Universal Robots PolyScope program: tip_change_JF.urp

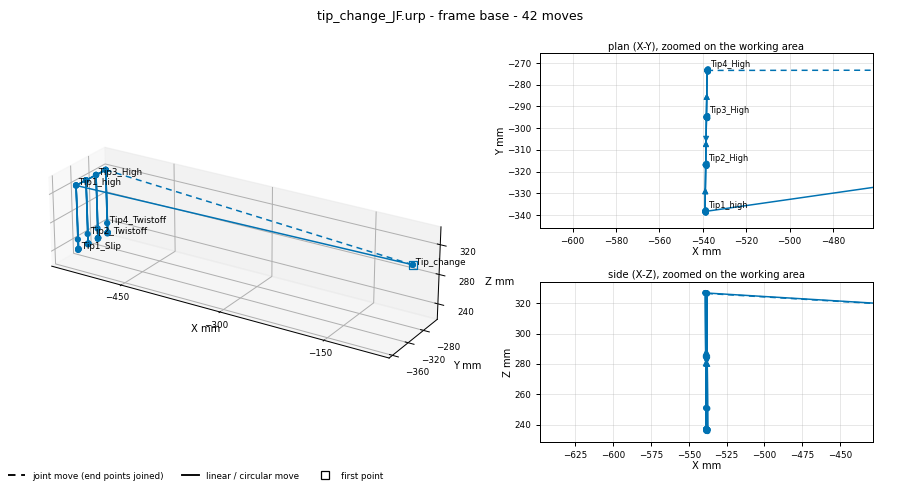
[picture p0: tool path of tip_change_JF.urp in frame base, 42 of 42 moves have a stored position in this frame; points joined in program order, loops and branches not executed]
Program tip_change_JF (installation=default directory=/programs/usbdisk/Ur-Program/Tip_change createdIn=3.10.1.76190 lastSavedIn=3.10.1.76190 robotSerialNumber=2018359886)
Calibrated DH parameters: a=[-0.000111, -0.180064, -0.391564, 0.000025, 0.000035, 0]; d=[0.089308, 162.079685, -160.155007, -1.814221, 0.094754, 0.082578]; alpha=[1.569707, -0.002379, 0.010338, 1.570474, -1.569894, 0]; deltaTheta=[0.000021, -1.133914, 1.184629, -0.050828, 0.000017, 0.000075]
Robot Program (runOnlyOnce=false)
  MoveJ speed 60 deg/s, acceleration 80 deg/s^2 (useActiveTCP=false) tcp=TCP_Tool1
    Waypoint Tip_change: TCP in base x=-81.571 y=-272.848 z=299.256 mm, rx=0 ry=0.0001 rz=-1.545 rad; joints [-70.556, -50.466, -101.854, -104.569, 84.569, 123.199] deg; flange x=-49.667 y=-215.719 z=542.134 mm, rx=2.3303 ry=1.8037 rz=-0.2542 rad
  Set NoAction tcp=TCP_Tool1
  'skipping tip 0-> No tool on robot'
  If Old_tip≟3
    MoveL speed 250 mm/s, acceleration 1200 mm/s^2 (useActiveTCP=false) tcp=TCP_Tool1; feature=Joint_6_name
      Waypoint Tip1_high: TCP in base x=-538.968 y=-338.378 z=326.942 mm, rx=-0.0068 ry=0.0085 rz=3.1265 rad; joints [-131.445, -107.957, -50.262, -104.103, 80.885, 154.293] deg; pose in feature x=57.214 y=-30.744 z=76.425 mm, rx=0 ry=0.0001 rz=-2.0641 rad; flange x=-490.354 y=-366.84 z=572.437 mm, rx=3.0721 ry=-0.4473 rz=-0.3327 rad
      Waypoint Tip1_Slip: TCP in base x=-538.568 y=-337.869 z=236.939 mm, rx=-0.0068 ry=0.0085 rz=3.1242 rad; joints [-131.488, -104.349, -68.619, -89.398, 80.899, 154.544] deg; pose in feature x=-140.414 y=-433.139 z=348.51 mm, rx=0.0255 ry=-0.0126 rz=-1.9429 rad; flange x=-490.024 y=-366.448 z=482.434 mm, rx=3.0718 ry=-0.4509 rz=-0.3328 rad
      Waypoint Tip1_Lock: TCP in base x=-538.583 y=-338.869 z=236.944 mm, rx=0.0013 ry=-0.0083 rz=-2.1118 rad; joints [-137.124, -99.221, -76.057, -82.468, 93.606, 89.965] deg; pose in feature x=-139.482 y=-433.5 z=348.531 mm, rx=0.0139 ry=-0.0208 rz=-0.8958 rad; flange x=-488.924 y=-309.541 z=482.128 mm, rx=2.7896 ry=1.107 rz=-0.2715 rad
      Waypoint Tip1_Twistoff: TCP in base x=-538.643 y=-338.793 z=250.944 mm, rx=-0.0027 ry=-0.0068 rz=-1.059 rad; joints [-143.816, -105.991, -63.242, -98.539, 103.242, 22.663] deg; pose in feature x=-0.02 y=-0.021 z=11.036 mm, rx=-0.0001 ry=0 rz=1.0527 rad; flange x=-538.901 y=-279.541 z=495.751 mm, rx=1.814 ry=2.3069 rz=-0.1444 rad
      Waypoint Tip1_high: TCP in base x=-538.968 y=-338.378 z=326.942 mm, rx=-0.0068 ry=0.0085 rz=3.1265 rad; joints [-131.445, -107.957, -50.262, -104.103, 80.885, 154.293] deg; pose in feature x=57.214 y=-30.744 z=76.425 mm, rx=0 ry=0.0001 rz=-2.0641 rad; flange x=-490.354 y=-366.84 z=572.437 mm, rx=3.0721 ry=-0.4473 rz=-0.3327 rad
    SuppressedNode
      MoveL speed 250 mm/s, acceleration 1200 mm/s^2 (useActiveTCP=false) tcp=TCP_Tool1; feature=Joint_6_name
        Waypoint Tip1_high: TCP in base x=-537.538 y=-337.809 z=326.901 mm, rx=0.0003 ry=0.0002 rz=-1.5826 rad; joints [-130.16, -106.928, -52.243, -102.922, -281.606, 155.501] deg; pose in feature x=0.604 y=0.279 z=0.912 mm, rx=0 ry=0.0001 rz=0.0099 rad; flange x=-481.613 y=-371.883 z=569.759 mm, rx=3.08 ry=-0.4512 rz=-0.394 rad
        Waypoint Tip1_press: TCP in base x=-537.53 y=-337.783 z=237.901 mm, rx=0.0003 ry=0 rz=-0.5354 rad; joints [-136.639, -97.589, -78.691, -79.527, -267.198, 90.394] deg; pose in feature x=-0.011 y=0.014 z=-89.017 mm, rx=0 ry=-0.0001 rz=1.0471 rad; flange x=-480.131 y=-306.405 z=480.779 mm, rx=2.7834 ry=1.1057 rz=-0.3248 rad
        Waypoint Tip1_Lock: TCP in base x=-537.531 y=-337.784 z=239.901 mm, rx=0.0003 ry=0 rz=-0.5354 rad; joints [-136.638, -97.608, -78.375, -79.823, -267.198, 90.392] deg; pose in feature x=-0.011 y=0.014 z=-87.017 mm, rx=0 ry=0 rz=1.0471 rad; flange x=-480.132 y=-306.408 z=482.779 mm, rx=2.7834 ry=1.1057 rz=-0.3248 rad
        Waypoint Tip1_Slip: TCP in base x=-537.531 y=-337.783 z=238.901 mm, rx=0.0003 ry=0.0001 rz=-1.5826 rad; joints [-130.205, -103.681, -69.728, -88.707, -281.576, 155.612] deg; pose in feature x=0.094 y=0.018 z=1.031 mm, rx=-0.0001 ry=-0.0001 rz=0.0001 rad; flange x=-481.61 y=-371.853 z=481.761 mm, rx=3.0799 ry=-0.4512 rz=-0.3939 rad
        Waypoint Tip1_high: TCP in base x=-537.538 y=-337.809 z=326.901 mm, rx=0.0003 ry=0.0002 rz=-1.5826 rad; joints [-130.16, -106.928, -52.243, -102.922, -281.606, 155.501] deg; pose in feature x=0.604 y=0.279 z=0.912 mm, rx=0 ry=0.0001 rz=0.0099 rad; flange x=-481.613 y=-371.883 z=569.759 mm, rx=3.08 ry=-0.4512 rz=-0.394 rad
  If Old_tip≟4
    MoveL speed 250 mm/s, acceleration 1200 mm/s^2 (useActiveTCP=false) tcp=TCP_Tool1; feature=Joint_6_name
      Waypoint Tip2_High: TCP in base x=-538.644 y=-316.88 z=326.826 mm, rx=-0.0068 ry=0.0085 rz=3.1265 rad; joints [-132.848, -105.784, -53.248, -103.06, 81.079, 152.898] deg; pose in feature x=2.19 y=1.693 z=81.747 mm, rx=-0.0035 ry=0.0068 rz=-0.958 rad; flange x=-490.029 y=-345.343 z=572.321 mm, rx=3.0721 ry=-0.4473 rz=-0.3327 rad
      Waypoint Tip2_Slip: TCP in base x=-538.244 y=-316.372 z=236.823 mm, rx=-0.0068 ry=0.0085 rz=3.1265 rad; joints [-132.898, -102.409, -71.128, -88.573, 81.109, 153.006] deg; pose in feature x=-160.454 y=-425.366 z=348.057 mm, rx=0.0255 ry=-0.0126 rz=-1.9406 rad; flange x=-489.629 y=-344.835 z=482.318 mm, rx=3.0721 ry=-0.4473 rz=-0.3327 rad
      Waypoint Tip2_Lock: TCP in base x=-538.259 y=-317.372 z=236.828 mm, rx=0.0012 ry=-0.0083 rz=-2.1095 rad; joints [-138.801, -97.64, -77.885, -82.321, 93.99, 88.197] deg; pose in feature x=-159.522 y=-425.727 z=348.078 mm, rx=0.0138 ry=-0.0208 rz=-0.8934 rad; flange x=-488.666 y=-287.924 z=482.011 mm, rx=2.7881 ry=1.1102 rz=-0.2712 rad
      Waypoint Tip2_Twistoff: TCP in base x=-538.319 y=-317.295 z=250.828 mm, rx=-0.0027 ry=-0.0068 rz=-1.0623 rad; joints [-145.487, -104.574, -65.006, -98.529, 103.298, 21.145] deg; pose in feature x=-0.013 y=0.071 z=-74.909 mm, rx=0.0001 ry=-0.0001 rz=2.0945 rad; flange x=-538.389 y=-258.046 z=495.635 mm, rx=1.8178 ry=2.3041 rz=-0.1448 rad
      Waypoint Tip2_High: TCP in base x=-538.644 y=-316.88 z=326.826 mm, rx=-0.0068 ry=0.0085 rz=3.1265 rad; joints [-132.848, -105.784, -53.248, -103.06, 81.079, 152.898] deg; pose in feature x=2.19 y=1.693 z=81.747 mm, rx=-0.0035 ry=0.0068 rz=-0.958 rad; flange x=-490.029 y=-345.343 z=572.321 mm, rx=3.0721 ry=-0.4473 rz=-0.3327 rad
    SuppressedNode
      MoveL speed 250 mm/s, acceleration 1200 mm/s^2 (useActiveTCP=false) tcp=TCP_Tool1; feature=Joint_6_name
        Waypoint Tip2_High: TCP in base x=-537.283 y=-316.311 z=326.907 mm, rx=0.0003 ry=0.0002 rz=-1.5826 rad; joints [-131.544, -104.755, -55.177, -101.873, -281.409, 154.115] deg; pose in feature x=-21.513 y=0.011 z=-0.018 mm, rx=0 ry=0 rz=-0.0001 rad; flange x=-481.359 y=-350.384 z=569.766 mm, rx=3.08 ry=-0.4512 rz=-0.394 rad
        Waypoint Tip2_Press: TCP in base x=-537.276 y=-316.285 z=237.907 mm, rx=0.0003 ry=0 rz=-0.5354 rad; joints [-138.326, -96.017, -80.448, -79.412, -266.784, 88.762] deg; pose in feature x=-21.511 y=0.015 z=-89.018 mm, rx=0 ry=-0.0001 rz=1.0471 rad; flange x=-479.877 y=-284.907 z=480.785 mm, rx=2.7834 ry=1.1057 rz=-0.3248 rad
        Waypoint Tip2_Lock: TCP in base x=-537.276 y=-316.285 z=239.907 mm, rx=0.0003 ry=0 rz=-0.5354 rad; joints [-138.325, -96.035, -80.135, -79.708, -266.784, 88.759] deg; pose in feature x=-21.511 y=0.015 z=-87.018 mm, rx=0 ry=0 rz=1.0471 rad; flange x=-479.878 y=-284.909 z=482.785 mm, rx=2.7834 ry=1.1057 rz=-0.3248 rad
        Waypoint Tip2_Slip: TCP in base x=-537.276 y=-316.285 z=238.907 mm, rx=0.0003 ry=0.0001 rz=-1.5826 rad; joints [-131.59, -101.734, -72.212, -87.881, -281.381, 154.223] deg; pose in feature x=-21.511 y=0.015 z=-88.018 mm, rx=0.0001 ry=0 rz=-0.0001 rad; flange x=-481.356 y=-350.354 z=481.767 mm, rx=3.0799 ry=-0.4512 rz=-0.3939 rad
        Waypoint Tip2_High: TCP in base x=-537.283 y=-316.311 z=326.907 mm, rx=0.0003 ry=0.0002 rz=-1.5826 rad; joints [-131.544, -104.755, -55.177, -101.873, -281.409, 154.115] deg; pose in feature x=-21.513 y=0.011 z=-0.018 mm, rx=0 ry=0 rz=-0.0001 rad; flange x=-481.359 y=-350.384 z=569.766 mm, rx=3.08 ry=-0.4512 rz=-0.394 rad
  If Old_tip≟5
    MoveL speed 250 mm/s, acceleration 1200 mm/s^2 (useActiveTCP=false) tcp=TCP_Tool1; feature=Joint_6_name
      Waypoint Tip3_High: TCP in base x=-538.312 y=-294.883 z=326.707 mm, rx=-0.0068 ry=0.0085 rz=3.1265 rad; joints [-134.359, -103.714, -56.012, -102.124, 81.293, 151.396] deg; pose in feature x=13.69 y=-3.755 z=-38.348 mm, rx=-0.1637 ry=0.1574 rz=-0.0025 rad; flange x=-489.697 y=-323.346 z=572.202 mm, rx=3.0721 ry=-0.4473 rz=-0.3327 rad
      Waypoint Tip3_Slip: TCP in base x=-537.912 y=-294.375 z=236.704 mm, rx=-0.0068 ry=0.0085 rz=3.1265 rad; joints [-134.411, -100.547, -73.471, -87.848, 81.321, 151.499] deg; pose in feature x=-180.961 y=-417.412 z=347.593 mm, rx=0.0255 ry=-0.0126 rz=-1.9406 rad; flange x=-489.297 y=-322.838 z=482.199 mm, rx=3.0721 ry=-0.4473 rz=-0.3327 rad
      Waypoint Tip3_Lock: TCP in base x=-537.927 y=-295.375 z=236.709 mm, rx=0.0012 ry=-0.0083 rz=-2.1095 rad; joints [-140.58, -96.119, -79.595, -82.242, 94.365, 86.458] deg; pose in feature x=-180.029 y=-417.773 z=347.614 mm, rx=0.0138 ry=-0.0208 rz=-0.8934 rad; flange x=-488.334 y=-265.927 z=481.892 mm, rx=2.7881 ry=1.1102 rz=-0.2712 rad
      Waypoint Tip3_Twistoff: TCP in base x=-537.987 y=-295.298 z=250.709 mm, rx=-0.0027 ry=-0.0068 rz=-1.0623 rad; joints [-147.274, -103.276, -66.568, -98.672, 103.353, 19.316] deg; pose in feature x=-1.767 y=-0.914 z=5.336 mm, rx=0 ry=0 rz=1.0005 rad; flange x=-538.057 y=-236.049 z=495.517 mm, rx=1.8178 ry=2.3041 rz=-0.1448 rad
      Waypoint Tip3_High: TCP in base x=-538.312 y=-294.883 z=326.707 mm, rx=-0.0068 ry=0.0085 rz=3.1265 rad; joints [-134.359, -103.714, -56.012, -102.124, 81.293, 151.396] deg; pose in feature x=13.69 y=-3.755 z=-38.348 mm, rx=-0.1637 ry=0.1574 rz=-0.0025 rad; flange x=-489.697 y=-323.346 z=572.202 mm, rx=3.0721 ry=-0.4473 rz=-0.3327 rad
    SuppressedNode
      MoveL speed 250 mm/s, acceleration 1200 mm/s^2 (useActiveTCP=false) tcp=TCP_Tool1; feature=Joint_6_name
        Waypoint Tip3_High: TCP in base x=-537.023 y=-294.313 z=326.914 mm, rx=0.0003 ry=0.0002 rz=-1.5826 rad; joints [-133.038, -102.675, -57.902, -100.922, -281.189, 152.62] deg; pose in feature x=-43.513 y=0.013 z=-0.018 mm, rx=0 ry=0 rz=-0.0001 rad; flange x=-481.098 y=-328.386 z=569.772 mm, rx=3.08 ry=-0.4512 rz=-0.394 rad
        Waypoint Tip3_Press: TCP in base x=-537.016 y=-294.286 z=237.914 mm, rx=0.0003 ry=0 rz=-0.5354 rad; joints [-140.139, -94.506, -82.089, -79.372, -266.341, 87.005] deg; pose in feature x=-43.511 y=0.017 z=-89.018 mm, rx=0 ry=-0.0001 rz=1.0471 rad; flange x=-479.616 y=-262.908 z=480.792 mm, rx=2.7834 ry=1.1057 rz=-0.3248 rad
        Waypoint Tip3_Lock: TCP in base x=-537.016 y=-294.287 z=239.914 mm, rx=0.0003 ry=0 rz=-0.5354 rad; joints [-140.138, -94.523, -81.777, -79.667, -266.341, 87.003] deg; pose in feature x=-43.511 y=0.016 z=-87.018 mm, rx=0 ry=0 rz=1.0471 rad; flange x=-479.617 y=-262.911 z=482.792 mm, rx=2.7834 ry=1.1057 rz=-0.3248 rad
        Waypoint Tip3_Slip: TCP in base x=-537.016 y=-294.286 z=238.914 mm, rx=0.0003 ry=0.0001 rz=-1.5826 rad; joints [-133.083, -99.839, -74.567, -87.115, -281.163, 152.725] deg; pose in feature x=-43.511 y=0.017 z=-88.018 mm, rx=0.0001 ry=0 rz=-0.0001 rad; flange x=-481.095 y=-328.356 z=481.774 mm, rx=3.0799 ry=-0.4512 rz=-0.3939 rad
        Waypoint Tip3_High: TCP in base x=-537.023 y=-294.313 z=326.914 mm, rx=0.0003 ry=0.0002 rz=-1.5826 rad; joints [-133.038, -102.675, -57.902, -100.922, -281.189, 152.62] deg; pose in feature x=-43.513 y=0.013 z=-0.018 mm, rx=0 ry=0 rz=-0.0001 rad; flange x=-481.098 y=-328.386 z=569.772 mm, rx=3.08 ry=-0.4512 rz=-0.394 rad
  If Old_tip≟6
    MoveL speed 250 mm/s, acceleration 1200 mm/s^2 (useActiveTCP=false) tcp=TCP_Tool1; feature=Joint_6_name
      Waypoint Tip4_High: TCP in base x=-537.988 y=-273.386 z=326.591 mm, rx=-0.0068 ry=0.0085 rz=3.1265 rad; joints [-135.913, -101.826, -58.462, -101.318, 81.519, 149.851] deg; pose in feature x=-0.038 y=0.033 z=76.429 mm, rx=0 ry=0.0001 rz=-2.0641 rad; flange x=-489.373 y=-301.849 z=572.086 mm, rx=3.0721 ry=-0.4473 rz=-0.3327 rad
      Waypoint Tip4_Slip: TCP in base x=-537.588 y=-272.878 z=236.588 mm, rx=-0.0068 ry=0.0085 rz=3.1265 rad; joints [-135.967, -98.824, -75.586, -87.211, 81.546, 149.951] deg; pose in feature x=-201.001 y=-409.638 z=347.14 mm, rx=0.0255 ry=-0.0126 rz=-1.9406 rad; flange x=-488.973 y=-301.34 z=482.083 mm, rx=3.0721 ry=-0.4473 rz=-0.3327 rad
      Waypoint Tip4_Lock: TCP in base x=-537.603 y=-273.877 z=236.593 mm, rx=0.0012 ry=-0.0083 rz=-2.1095 rad; joints [-142.401, -94.732, -81.112, -82.237, 94.745, 84.676] deg; pose in feature x=-200.069 y=-410 z=347.161 mm, rx=0.0138 ry=-0.0208 rz=-0.8934 rad; flange x=-488.01 y=-244.43 z=481.776 mm, rx=2.7881 ry=1.1102 rz=-0.2712 rad
      Waypoint Tip4_Twistoff: TCP in base x=-537.663 y=-273.801 z=250.593 mm, rx=-0.0027 ry=-0.0068 rz=-1.0623 rad; joints [-149.082, -102.119, -67.921, -98.888, 103.396, 17.462] deg; pose in feature x=-0.04 y=0.039 z=0.429 mm, rx=0.0001 ry=0 rz=0.0303 rad; flange x=-537.733 y=-214.552 z=495.401 mm, rx=1.8178 ry=2.3041 rz=-0.1448 rad
      Waypoint Tip4_High: TCP in base x=-537.988 y=-273.386 z=326.591 mm, rx=-0.0068 ry=0.0085 rz=3.1265 rad; joints [-135.913, -101.826, -58.462, -101.318, 81.519, 149.851] deg; pose in feature x=-0.038 y=0.033 z=76.429 mm, rx=0 ry=0.0001 rz=-2.0641 rad; flange x=-489.373 y=-301.849 z=572.086 mm, rx=3.0721 ry=-0.4473 rz=-0.3327 rad
    SuppressedNode
      MoveL speed 250 mm/s, acceleration 1200 mm/s^2 (useActiveTCP=false) tcp=TCP_Tool1; feature=Joint_6_name
        Waypoint Tip4_High: TCP in base x=-536.768 y=-272.814 z=326.92 mm, rx=0.0003 ry=0.0002 rz=-1.5826 rad; joints [-134.575, -100.773, -60.327, -100.092, -280.955, 151.081] deg; pose in feature x=-65.013 y=0.014 z=-0.019 mm, rx=0 ry=0 rz=-0.0001 rad; flange x=-480.844 y=-306.888 z=569.779 mm, rx=3.08 ry=-0.4512 rz=-0.394 rad
        Waypoint Tip4_Press: TCP in base x=-536.761 y=-272.788 z=237.92 mm, rx=0.0003 ry=0 rz=-0.5354 rad; joints [-141.998, -93.127, -83.542, -79.403, -265.89, 85.201] deg; pose in feature x=-65.011 y=0.018 z=-89.019 mm, rx=0 ry=-0.0001 rz=1.0471 rad; flange x=-479.362 y=-241.41 z=480.798 mm, rx=2.7834 ry=1.1057 rz=-0.3248 rad
        Waypoint Tip4_Lock: TCP in base x=-536.761 y=-272.788 z=239.92 mm, rx=0.0003 ry=0 rz=-0.5354 rad; joints [-141.997, -93.144, -83.231, -79.697, -265.89, 85.199] deg; pose in feature x=-65.011 y=0.018 z=-87.019 mm, rx=0 ry=0 rz=1.0471 rad; flange x=-479.363 y=-241.412 z=482.798 mm, rx=2.7834 ry=1.1057 rz=-0.3248 rad
        Waypoint Tip4_Slip: TCP in base x=-536.761 y=-272.788 z=238.92 mm, rx=0.0003 ry=0.0001 rz=-1.5826 rad; joints [-134.621, -98.08, -76.697, -86.434, -280.931, 151.185] deg; pose in feature x=-65.011 y=0.018 z=-88.019 mm, rx=0.0001 ry=0 rz=-0.0001 rad; flange x=-480.841 y=-306.857 z=481.78 mm, rx=3.0799 ry=-0.4512 rz=-0.3939 rad
        Waypoint Tip4_High: TCP in base x=-536.768 y=-272.814 z=326.92 mm, rx=0.0003 ry=0.0002 rz=-1.5826 rad; joints [-134.575, -100.773, -60.327, -100.092, -280.955, 151.081] deg; pose in feature x=-65.013 y=0.014 z=-0.019 mm, rx=0 ry=0 rz=-0.0001 rad; flange x=-480.844 y=-306.888 z=569.779 mm, rx=3.08 ry=-0.4512 rz=-0.394 rad
  If New_tip≟3
    MoveL speed 250 mm/s, acceleration 1200 mm/s^2 (useActiveTCP=false) tcp=TCP_Tool1; feature=Joint_6_name
      Waypoint Tip1_high: TCP in base x=-538.968 y=-338.378 z=326.942 mm, rx=-0.0068 ry=0.0085 rz=3.1265 rad; joints [-131.445, -107.957, -50.262, -104.103, 80.885, 154.293] deg; pose in feature x=57.214 y=-30.744 z=76.425 mm, rx=0 ry=0.0001 rz=-2.0641 rad; flange x=-490.354 y=-366.84 z=572.437 mm, rx=3.0721 ry=-0.4473 rz=-0.3327 rad
      Waypoint Tip1_press: TCP in base x=-538.579 y=-338.875 z=235.944 mm, rx=0.0013 ry=-0.0083 rz=-2.1118 rad; joints [-137.124, -99.209, -76.218, -82.319, 93.606, 89.967] deg; pose in feature x=-139.458 y=-433.497 z=347.532 mm, rx=0.0139 ry=-0.0208 rz=-0.8958 rad; flange x=-488.92 y=-309.546 z=481.128 mm, rx=2.7896 ry=1.107 rz=-0.2715 rad
      Waypoint Tip1_Lock: TCP in base x=-538.583 y=-338.869 z=236.944 mm, rx=0.0013 ry=-0.0083 rz=-2.1118 rad; joints [-137.124, -99.221, -76.057, -82.468, 93.606, 89.965] deg; pose in feature x=-139.482 y=-433.5 z=348.531 mm, rx=0.0139 ry=-0.0208 rz=-0.8958 rad; flange x=-488.924 y=-309.541 z=482.128 mm, rx=2.7896 ry=1.107 rz=-0.2715 rad
      Waypoint Tip1_Slip: TCP in base x=-538.568 y=-337.869 z=236.939 mm, rx=-0.0068 ry=0.0085 rz=3.1242 rad; joints [-131.488, -104.349, -68.619, -89.398, 80.899, 154.544] deg; pose in feature x=-140.414 y=-433.139 z=348.51 mm, rx=0.0255 ry=-0.0126 rz=-1.9429 rad; flange x=-490.024 y=-366.448 z=482.434 mm, rx=3.0718 ry=-0.4509 rz=-0.3328 rad
      Waypoint Tip1_high: TCP in base x=-538.968 y=-338.378 z=326.942 mm, rx=-0.0068 ry=0.0085 rz=3.1265 rad; joints [-131.445, -107.957, -50.262, -104.103, 80.885, 154.293] deg; pose in feature x=57.214 y=-30.744 z=76.425 mm, rx=0 ry=0.0001 rz=-2.0641 rad; flange x=-490.354 y=-366.84 z=572.437 mm, rx=3.0721 ry=-0.4473 rz=-0.3327 rad
  If New_tip≟4
    MoveL speed 250 mm/s, acceleration 1200 mm/s^2 (useActiveTCP=false) tcp=TCP_Tool1; feature=Joint_6_name
      Waypoint Tip2_High: TCP in base x=-538.644 y=-316.88 z=326.826 mm, rx=-0.0068 ry=0.0085 rz=3.1265 rad; joints [-132.848, -105.784, -53.248, -103.06, 81.079, 152.898] deg; pose in feature x=2.19 y=1.693 z=81.747 mm, rx=-0.0035 ry=0.0068 rz=-0.958 rad; flange x=-490.029 y=-345.343 z=572.321 mm, rx=3.0721 ry=-0.4473 rz=-0.3327 rad
      Waypoint Tip2_Press: TCP in base x=-538.255 y=-317.377 z=235.828 mm, rx=0.0012 ry=-0.0083 rz=-2.1095 rad; joints [-138.8, -97.629, -78.044, -82.173, 93.99, 88.199] deg; pose in feature x=-159.498 y=-425.724 z=347.078 mm, rx=0.0138 ry=-0.0208 rz=-0.8934 rad; flange x=-488.662 y=-287.93 z=481.011 mm, rx=2.7881 ry=1.1102 rz=-0.2712 rad
      Waypoint Tip2_Lock: TCP in base x=-538.259 y=-317.372 z=236.828 mm, rx=0.0012 ry=-0.0083 rz=-2.1095 rad; joints [-138.801, -97.64, -77.885, -82.321, 93.99, 88.197] deg; pose in feature x=-159.522 y=-425.727 z=348.078 mm, rx=0.0138 ry=-0.0208 rz=-0.8934 rad; flange x=-488.666 y=-287.924 z=482.011 mm, rx=2.7881 ry=1.1102 rz=-0.2712 rad
      Waypoint Tip2_Slip: TCP in base x=-538.244 y=-316.372 z=236.823 mm, rx=-0.0068 ry=0.0085 rz=3.1265 rad; joints [-132.898, -102.409, -71.128, -88.573, 81.109, 153.006] deg; pose in feature x=-160.454 y=-425.366 z=348.057 mm, rx=0.0255 ry=-0.0126 rz=-1.9406 rad; flange x=-489.629 y=-344.835 z=482.318 mm, rx=3.0721 ry=-0.4473 rz=-0.3327 rad
      Waypoint Tip2_High: TCP in base x=-538.644 y=-316.88 z=326.826 mm, rx=-0.0068 ry=0.0085 rz=3.1265 rad; joints [-132.848, -105.784, -53.248, -103.06, 81.079, 152.898] deg; pose in feature x=2.19 y=1.693 z=81.747 mm, rx=-0.0035 ry=0.0068 rz=-0.958 rad; flange x=-490.029 y=-345.343 z=572.321 mm, rx=3.0721 ry=-0.4473 rz=-0.3327 rad
  If New_tip≟5
    MoveL speed 250 mm/s, acceleration 1200 mm/s^2 (useActiveTCP=false) tcp=TCP_Tool1; feature=Joint_6_name
      Waypoint Tip3_High: TCP in base x=-538.312 y=-294.883 z=326.707 mm, rx=-0.0068 ry=0.0085 rz=3.1265 rad; joints [-134.359, -103.714, -56.012, -102.124, 81.293, 151.396] deg; pose in feature x=13.69 y=-3.755 z=-38.348 mm, rx=-0.1637 ry=0.1574 rz=-0.0025 rad; flange x=-489.697 y=-323.346 z=572.202 mm, rx=3.0721 ry=-0.4473 rz=-0.3327 rad
      Waypoint Tip3_Press: TCP in base x=-537.923 y=-295.38 z=235.709 mm, rx=0.0012 ry=-0.0083 rz=-2.1095 rad; joints [-140.579, -96.109, -79.753, -82.094, 94.365, 86.46] deg; pose in feature x=-180.005 y=-417.77 z=346.615 mm, rx=0.0138 ry=-0.0208 rz=-0.8934 rad; flange x=-488.33 y=-265.932 z=480.892 mm, rx=2.7881 ry=1.1102 rz=-0.2712 rad
      Waypoint Tip3_Lock: TCP in base x=-537.927 y=-295.375 z=236.709 mm, rx=0.0012 ry=-0.0083 rz=-2.1095 rad; joints [-140.58, -96.119, -79.595, -82.242, 94.365, 86.458] deg; pose in feature x=-180.029 y=-417.773 z=347.614 mm, rx=0.0138 ry=-0.0208 rz=-0.8934 rad; flange x=-488.334 y=-265.927 z=481.892 mm, rx=2.7881 ry=1.1102 rz=-0.2712 rad
      Waypoint Tip3_Slip: TCP in base x=-537.912 y=-294.375 z=236.704 mm, rx=-0.0068 ry=0.0085 rz=3.1265 rad; joints [-134.411, -100.547, -73.471, -87.848, 81.321, 151.499] deg; pose in feature x=-180.961 y=-417.412 z=347.593 mm, rx=0.0255 ry=-0.0126 rz=-1.9406 rad; flange x=-489.297 y=-322.838 z=482.199 mm, rx=3.0721 ry=-0.4473 rz=-0.3327 rad
      Waypoint Tip3_High: TCP in base x=-538.312 y=-294.883 z=326.707 mm, rx=-0.0068 ry=0.0085 rz=3.1265 rad; joints [-134.359, -103.714, -56.012, -102.124, 81.293, 151.396] deg; pose in feature x=13.69 y=-3.755 z=-38.348 mm, rx=-0.1637 ry=0.1574 rz=-0.0025 rad; flange x=-489.697 y=-323.346 z=572.202 mm, rx=3.0721 ry=-0.4473 rz=-0.3327 rad
  If New_tip≟6
    MoveL speed 250 mm/s, acceleration 1200 mm/s^2 (useActiveTCP=false) tcp=TCP_Tool1; feature=Joint_6_name
      Waypoint Tip4_High: TCP in base x=-537.988 y=-273.386 z=326.591 mm, rx=-0.0068 ry=0.0085 rz=3.1265 rad; joints [-135.913, -101.826, -58.462, -101.318, 81.519, 149.851] deg; pose in feature x=-0.038 y=0.033 z=76.429 mm, rx=0 ry=0.0001 rz=-2.0641 rad; flange x=-489.373 y=-301.849 z=572.086 mm, rx=3.0721 ry=-0.4473 rz=-0.3327 rad
      Waypoint Tip4_Press: TCP in base x=-537.598 y=-273.883 z=235.593 mm, rx=0.0012 ry=-0.0083 rz=-2.1095 rad; joints [-142.401, -94.722, -81.27, -82.089, 94.744, 84.678] deg; pose in feature x=-200.045 y=-409.997 z=346.162 mm, rx=0.0138 ry=-0.0208 rz=-0.8934 rad; flange x=-488.005 y=-244.435 z=480.776 mm, rx=2.7881 ry=1.1102 rz=-0.2712 rad
      Waypoint Tip4_Lock: TCP in base x=-537.603 y=-273.877 z=236.593 mm, rx=0.0012 ry=-0.0083 rz=-2.1095 rad; joints [-142.401, -94.732, -81.112, -82.237, 94.745, 84.676] deg; pose in feature x=-200.069 y=-410 z=347.161 mm, rx=0.0138 ry=-0.0208 rz=-0.8934 rad; flange x=-488.01 y=-244.43 z=481.776 mm, rx=2.7881 ry=1.1102 rz=-0.2712 rad
      Waypoint Tip4_Slip: TCP in base x=-537.588 y=-272.878 z=236.588 mm, rx=-0.0068 ry=0.0085 rz=3.1265 rad; joints [-135.967, -98.824, -75.586, -87.211, 81.546, 149.951] deg; pose in feature x=-201.001 y=-409.638 z=347.14 mm, rx=0.0255 ry=-0.0126 rz=-1.9406 rad; flange x=-488.973 y=-301.34 z=482.083 mm, rx=3.0721 ry=-0.4473 rz=-0.3327 rad
      Waypoint Tip4_High: TCP in base x=-537.988 y=-273.386 z=326.591 mm, rx=-0.0068 ry=0.0085 rz=3.1265 rad; joints [-135.913, -101.826, -58.462, -101.318, 81.519, 149.851] deg; pose in feature x=-0.038 y=0.033 z=76.429 mm, rx=0 ry=0.0001 rz=-2.0641 rad; flange x=-489.373 y=-301.849 z=572.086 mm, rx=3.0721 ry=-0.4473 rz=-0.3327 rad
  MoveJ speed 60 deg/s, acceleration 80 deg/s^2 (useActiveTCP=false) tcp=TCP_Tool1
    Waypoint Tip_change: TCP in base x=-81.571 y=-272.848 z=299.256 mm, rx=0 ry=0.0001 rz=-1.545 rad; joints [-70.556, -50.466, -101.854, -104.569, 84.569, 123.199] deg; flange x=-49.667 y=-215.719 z=542.134 mm, rx=2.3303 ry=1.8037 rz=-0.2542 rad
  If New_tip≠0
    Set NoAction tcp=TCP_Tips
  Old_tip := New_tip
